INTERFACE I_AnalogInput EXTENDS I_Component, I_ForcibleInt

{attribute 'monitoring' := 'call'}
PROPERTY RawValue : INT
GET
END_GET
END_PROPERTY

{attribute 'monitoring' := 'call'}
PROPERTY Value : LREAL
GET
END_GET
END_PROPERTY

END_INTERFACE

(* stored: Version 1.1.0.1, ProductVersion 3.1.4026.18
   Itf I_AnalogInput: Id {ca0b1ff8-0439-4c6e-8139-d5055573ab0a}
   Property RawValue: Id {b67cacb0-5c45-4b1e-82d2-17a7d4adead9}
   Get Get: Id {f2731e27-7d6c-47d0-a64e-c485228eeaa4}
   Property Value: Id {3350fce4-1a93-4330-9a3e-79984e81f6ee}
   Get Get: Id {281b6989-3bcd-45cb-accf-8a98952f4483} *)
